Universal Robots PolyScope program: programa2.urp

Program programa2 (installation=default directory=/ursim/programs createdIn=5.26.1 lastSavedIn=5.26.1 robotSerialNumber=20195599999)
Calibrated DH parameters: a=[0, -0.425, -0.3922, 0, 0, 0]; d=[0.1625, 0, 0, 0.1333, 0.0997, 0.0996]; alpha=[1.570796, 0, 0, 1.570796, -1.570796, 0]; deltaTheta=[0, 0, 0, 0, 0, 0]
InitVariablesNode
Robot Program (runOnlyOnce=false)
  Set DigitalOutput pin=digital_out[0]; digitalValue=1
  Popup Message (haltProgram=false message=el control va a ser compartido con un controlador externo inputType=Text)
  Wait Sleep waitTime=5
  URCap External Control (External Control, FZI Research Center for Information Technology)
